TYPE Tag_UID : ARRAY[0..7] OF USINT; END_TYPE

(* stored: Version 1.1.0.1, ProductVersion 3.1.4024.10
   DUT Tag_UID: Id {eeeac8b5-fdc9-4396-8f23-d16d4757bda2} *)
